{attribute 'linkalways'} 
{attribute 'no_explicit_call' := 'This FB is a CLASS and must be accessed using methods or properties'}
{attribute 'enable_dynamic_creation'}
FUNCTION_BLOCK _DT EXTENDS DatatypeBase
VAR
	localData : DT;
	activeData : REFERENCE TO DT REF= localData;
END_VAR

PROPERTY PUBLIC Address : PVOID
GET
Address := ADR(activeData);
END_GET
END_PROPERTY

METHOD PUBLIC ClearReference
VAR_INPUT
END_VAR
activeData REF= localData;
END_METHOD

METHOD PUBLIC Clone : I_Datatype
VAR
    pClone : POINTER TO _DT;
END_VAR
pClone := __NEW(_DT(InitialValue := Value));
Clone := pClone^;
END_METHOD

METHOD FB_init : BOOL
VAR_INPUT
	bInitRetains : BOOL; // if TRUE, the retain variables are initialized (warm start / cold start)
	bInCopyCode : BOOL;  // if TRUE, the instance afterwards gets moved WORDo the copy code (online change)
	InitialValue : DT;
END_VAR
localData := InitialValue;
END_METHOD

METHOD PUBLIC MakeReferenceTo
VAR_INPUT
	ReferenceTarget : REFERENCE TO DT;
END_VAR
activeData REF= ReferenceTarget;
END_METHOD

METHOD PUBLIC SerializeWith
VAR_INPUT
	Serializer : I_Serializer;
END_VAR
Serializer.AddDateTime(activeData);
END_METHOD

PROPERTY PUBLIC Size : UDINT
GET
Size := SIZEOF(activeData);
END_GET
END_PROPERTY

METHOD TryDeserializeFrom : BOOL
VAR_INPUT
	Deserializer : I_Deserializer;
	Feedback : I_DeserializerFeedback;
END_VAR
TryDeserializeFrom := Deserializer.TryGetDateTime(activeData, Feedback);
END_METHOD

METHOD TryMakeReferenceTo : BOOL
VAR_INPUT
	Target : I_Datatype;
END_VAR
VAR
	pTargetData : POINTER TO DT;
END_VAR
IF NOT IsEquivalentTo(Target) THEN
	RETURN;
END_IF

pTargetData := Target.Address;
activeData REF= pTargetData^;
TryMakeReferenceTo := TRUE;
END_METHOD

PROPERTY PUBLIC TypeName : T_MAXSTRING
GET
TypeName := 'DT';
END_GET
END_PROPERTY

PROPERTY PUBLIC Value : REFERENCE TO DT
GET
Value REF= activeData;
END_GET
END_PROPERTY

END_FUNCTION_BLOCK

(* stored: Version 1.1.0.1, ProductVersion 3.1.4024.13
   POU _DT: Id {557fbd08-78d2-4290-a0a2-96907ad466de}, SpecialFunc None
   Folder Constructor: Id {1daddea9-d910-426e-98b0-518002b00b4f}
   Property Address: Id {f727ff13-6d02-4c69-8506-4cb70ca2a7b0}
   Get Get: Id {9b37e431-d915-4088-9a1a-ec542408e232}
   Method ClearReference: Id {7a899d5d-7c19-4ddf-ab52-cbcdc975db9d}
   Method Clone: Id {25f47063-836b-46ac-a729-5492e3e84eda}
   Method FB_init: Id {bbd765fa-5a03-4ea1-991a-2a98716134b9}
   Method MakeReferenceTo: Id {71982807-5509-478b-b50d-5a09b075de43}
   Method SerializeWith: Id {6fff3e7c-1041-468f-952d-3261c5f66b56}
   Property Size: Id {bf63aea1-4b92-4159-a201-703e6e2e6394}
   Get Get: Id {6e64fa1f-c505-4c83-b82e-eced92d1e0a2}
   Method TryDeserializeFrom: Id {474ea195-9ecc-42e0-ad4c-61dca0928d66}
   Method TryMakeReferenceTo: Id {723b503d-4198-4672-b636-df8de3af8a14}
   Property TypeName: Id {b6b24220-1a0b-491a-ae9f-daa860acd777}
   Get Get: Id {afae55cd-8070-4d6d-926f-5cdfe879b297}
   Property Value: Id {31c62ec5-0c35-4115-a7fc-233352071ea5}
   Get Get: Id {74af408e-40d0-46ed-8270-933717a9429c} *)
